(* Logix 5000 project; controller Drives_Line1 1756-L72 rev 20.13; software revision 20.04; part 10 of 21 *)
(* tags used below, declared in another part *)
   Bridle_01_FB_Count_Old : DINT;
   Bridle_01_Max_FBcounts : REAL;
   Bridle_01_SpdTrimMPS : REAL;
   Bridle_01_SpdTrimPct : REAL;
   Bridle_01a_RPMPerMPS : REAL;
   Bridle_01b_RPMPerMPS : REAL;
   Bridle_01c_RPMPerMPS : REAL;
   IO_State_Bridle_01a : INT;
   IO_State_Bridle_01b : INT;
   IO_State_Bridle_01c : INT;
   IO_State_Tmp_Bridle_01a : INT;
   IO_State_Tmp_Bridle_01b : INT;
   IO_State_Tmp_Bridle_01c : INT;
   zBridle_01_Ki_SpdTrim : REAL;
   zBridle_01_Kp_SpdTrim : REAL;
   zBridle_01_Max_rev : DINT;
   zBridle_01_MaxTrimSpdTrim : REAL;
   zBridle_01_MinTrimSpdTrim : REAL;
   zBridle_01b_EncRes : REAL;
   Bridle_01 : UDT_Bridle_3M;
   Bridle_01_FB_Diff : REAL;
   Bridle_01_FB_Update_Valid : BOOL;
   Bridle_01_Rev_mm : REAL;
   Bridle_01b_FBCounts_mm : REAL;
   EntryCtrl : UDT_Control_Zone;
   EntryStat : UDT_Status_Zone;
   LineCmd : UDT_Commands_Line;
   offst_pr_br1 : REAL;
   Out_Feedbacks : UDT_Fdbks;
   Out_Status : UDT_Status;
   TaskInterval_ms : DINT;
   TestConfig_Bridle_01a : UDT_Config_Bridle;
   TestConfig_Bridle_01b : UDT_Config_Bridle;
   TestConfig_Bridle_01c : UDT_Config_Bridle;
   voirmw : BOOL;
   zConfigFromMaster : BOOL;
   zPi : REAL;
   zSimulation : BOOL;
(* P14_Bridle_01, continued *)

ROUTINE R03_Drive_Interface   (* ladder *)
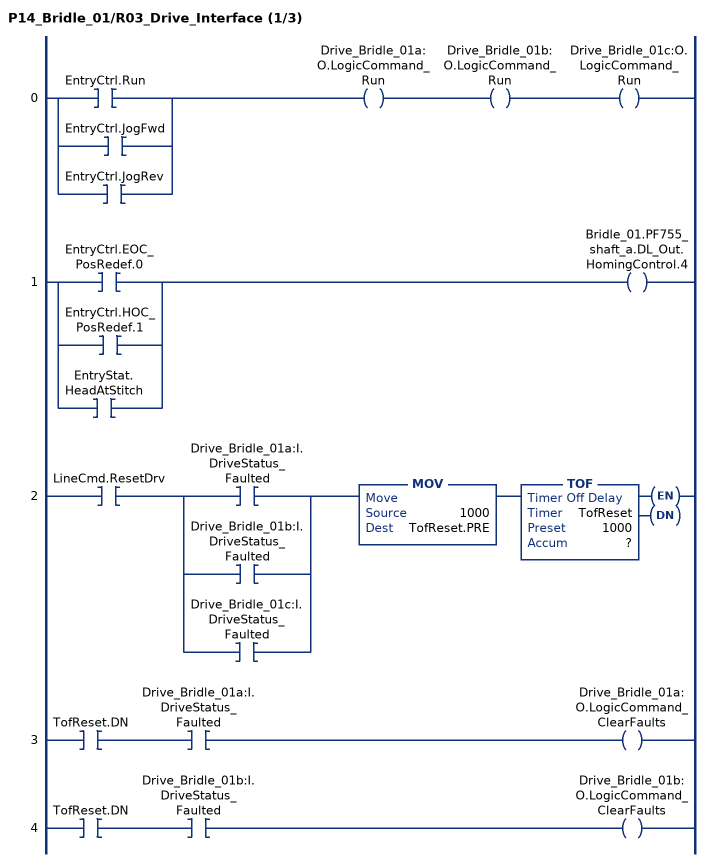
   0: [XIC(EntryCtrl.Run) ,XIC(EntryCtrl.JogFwd) ,XIC(EntryCtrl.JogRev) ]OTE(Drive_Bridle_01a:O.LogicCommand_Run)OTE(Drive_Bridle_01b:O.LogicCommand_Run)OTE(Drive_Bridle_01c:O.LogicCommand_Run);
   1: [XIC(EntryCtrl.EOC_PosRedef.0) ,XIC(EntryCtrl.HOC_PosRedef.1) ,XIC(EntryStat.HeadAtStitch) ]OTE(Bridle_01.PF755_shaft_a.DL_Out.HomingControl.4);
   2: XIC(LineCmd.ResetDrv)[XIC(Drive_Bridle_01a:I.DriveStatus_Faulted) ,XIC(Drive_Bridle_01b:I.DriveStatus_Faulted) ,XIC(Drive_Bridle_01c:I.DriveStatus_Faulted) ]MOV(1000,TofReset.PRE)TOF(TofReset,?,?);
   3: XIC(TofReset.DN)XIC(Drive_Bridle_01a:I.DriveStatus_Faulted)OTE(Drive_Bridle_01a:O.LogicCommand_ClearFaults);
   4: XIC(TofReset.DN)XIC(Drive_Bridle_01b:I.DriveStatus_Faulted)OTE(Drive_Bridle_01b:O.LogicCommand_ClearFaults);
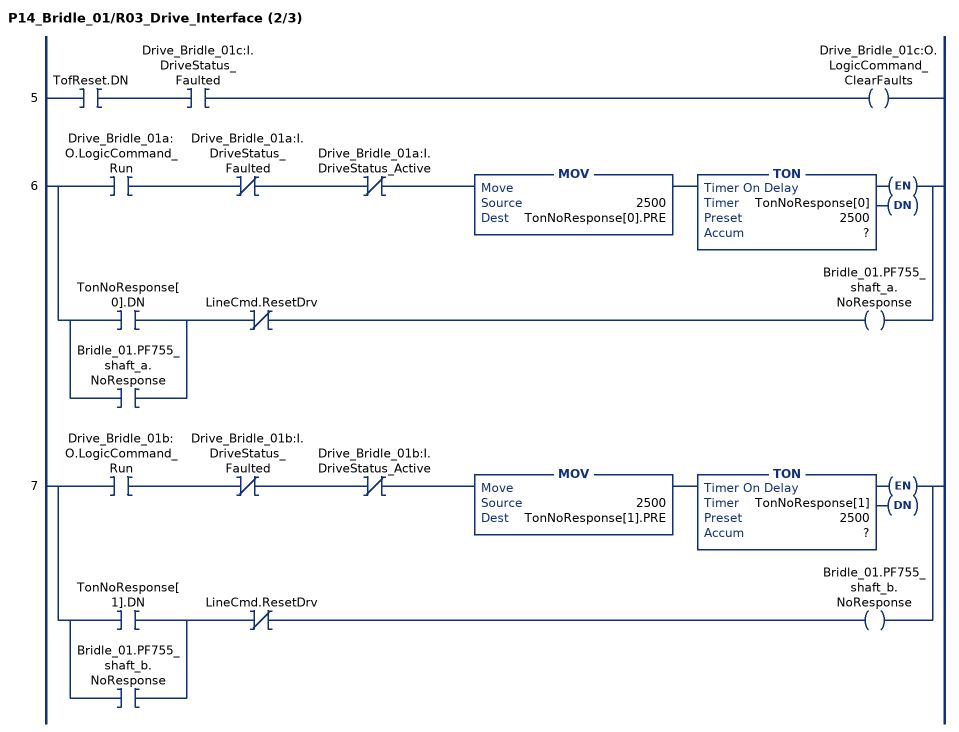
   5: XIC(TofReset.DN)XIC(Drive_Bridle_01c:I.DriveStatus_Faulted)OTE(Drive_Bridle_01c:O.LogicCommand_ClearFaults);
   6: [XIC(Drive_Bridle_01a:O.LogicCommand_Run) XIO(Drive_Bridle_01a:I.DriveStatus_Faulted) XIO(Drive_Bridle_01a:I.DriveStatus_Active) MOV(2500,TonNoResponse[0].PRE) TON(TonNoResponse[0],?,?) ,[XIC(TonNoResponse[0].DN) ,XIC(Bridle_01.PF755_shaft_a.NoResponse) ] XIO(LineCmd.ResetDrv) OTE(Bridle_01.PF755_shaft_a.NoResponse) ];
   7: [XIC(Drive_Bridle_01b:O.LogicCommand_Run) XIO(Drive_Bridle_01b:I.DriveStatus_Faulted) XIO(Drive_Bridle_01b:I.DriveStatus_Active) MOV(2500,TonNoResponse[1].PRE) TON(TonNoResponse[1],?,?) ,[XIC(TonNoResponse[1].DN) ,XIC(Bridle_01.PF755_shaft_b.NoResponse) ] XIO(LineCmd.ResetDrv) OTE(Bridle_01.PF755_shaft_b.NoResponse) ];
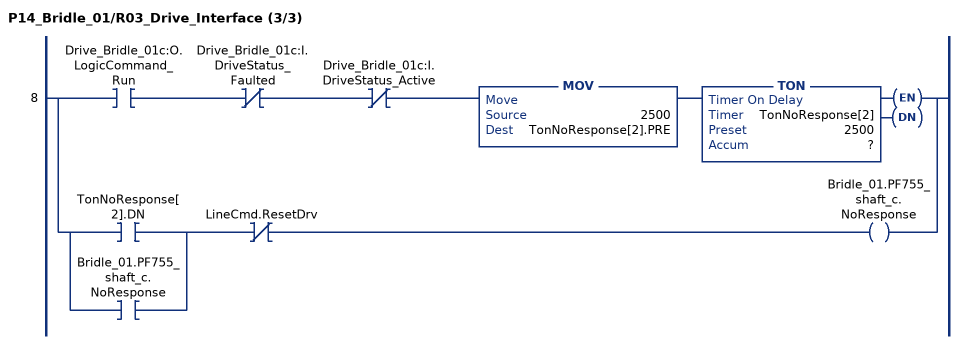
   8: [XIC(Drive_Bridle_01c:O.LogicCommand_Run) XIO(Drive_Bridle_01c:I.DriveStatus_Faulted) XIO(Drive_Bridle_01c:I.DriveStatus_Active) MOV(2500,TonNoResponse[2].PRE) TON(TonNoResponse[2],?,?) ,[XIC(TonNoResponse[2].DN) ,XIC(Bridle_01.PF755_shaft_c.NoResponse) ] XIO(LineCmd.ResetDrv) OTE(Bridle_01.PF755_shaft_c.NoResponse) ];
END_ROUTINE

ROUTINE R04_State   (* ladder *)
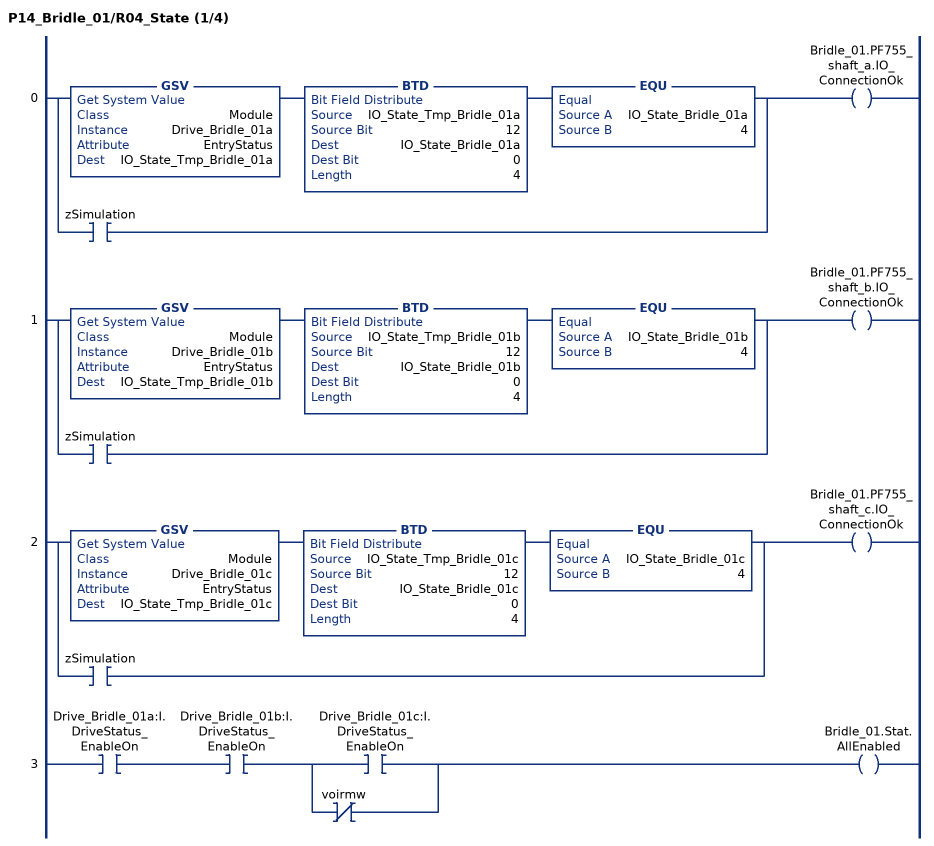
   0: [GSV(Module,Drive_Bridle_01a,EntryStatus,IO_State_Tmp_Bridle_01a) BTD(IO_State_Tmp_Bridle_01a,12,IO_State_Bridle_01a,0,4) EQU(IO_State_Bridle_01a,4) ,XIC(zSimulation) ]OTE(Bridle_01.PF755_shaft_a.IO_ConnectionOk);
   1: [GSV(Module,Drive_Bridle_01b,EntryStatus,IO_State_Tmp_Bridle_01b) BTD(IO_State_Tmp_Bridle_01b,12,IO_State_Bridle_01b,0,4) EQU(IO_State_Bridle_01b,4) ,XIC(zSimulation) ]OTE(Bridle_01.PF755_shaft_b.IO_ConnectionOk);
   2: [GSV(Module,Drive_Bridle_01c,EntryStatus,IO_State_Tmp_Bridle_01c) BTD(IO_State_Tmp_Bridle_01c,12,IO_State_Bridle_01c,0,4) EQU(IO_State_Bridle_01c,4) ,XIC(zSimulation) ]OTE(Bridle_01.PF755_shaft_c.IO_ConnectionOk);
   3: XIC(Drive_Bridle_01a:I.DriveStatus_EnableOn)XIC(Drive_Bridle_01b:I.DriveStatus_EnableOn)[XIC(Drive_Bridle_01c:I.DriveStatus_EnableOn) ,XIO(voirmw) ]OTE(Bridle_01.Stat.AllEnabled);
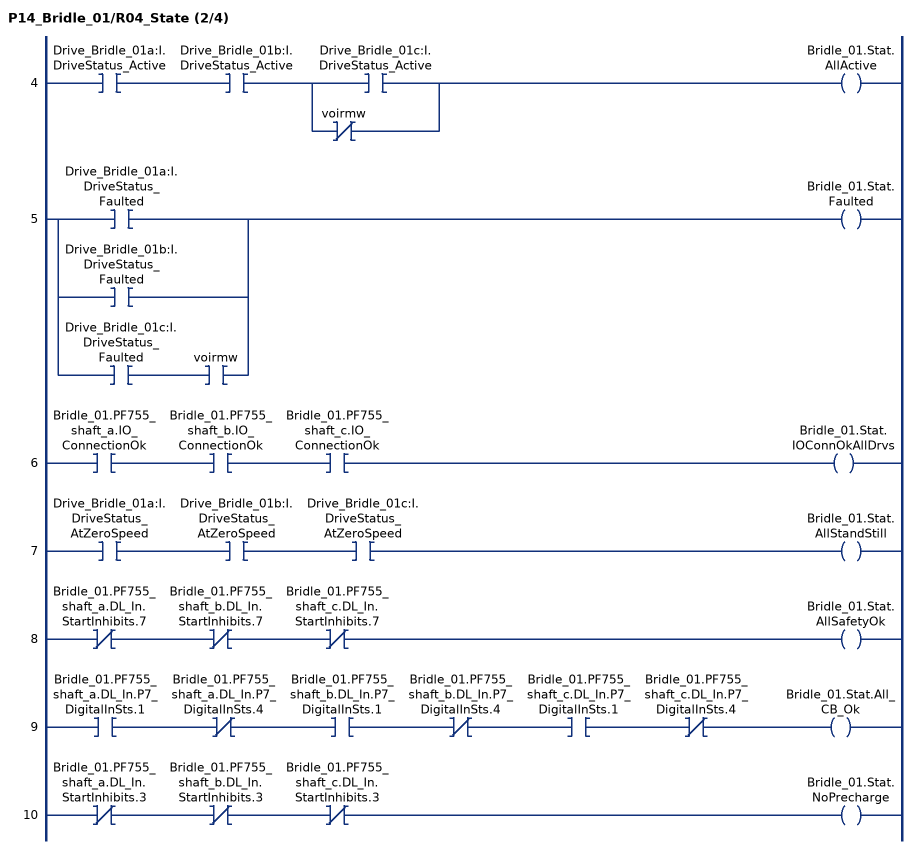
   4: XIC(Drive_Bridle_01a:I.DriveStatus_Active)XIC(Drive_Bridle_01b:I.DriveStatus_Active)[XIC(Drive_Bridle_01c:I.DriveStatus_Active) ,XIO(voirmw) ]OTE(Bridle_01.Stat.AllActive);
   5: [XIC(Drive_Bridle_01a:I.DriveStatus_Faulted) ,XIC(Drive_Bridle_01b:I.DriveStatus_Faulted) ,XIC(Drive_Bridle_01c:I.DriveStatus_Faulted) XIC(voirmw) ]OTE(Bridle_01.Stat.Faulted);
   6: XIC(Bridle_01.PF755_shaft_a.IO_ConnectionOk)XIC(Bridle_01.PF755_shaft_b.IO_ConnectionOk)XIC(Bridle_01.PF755_shaft_c.IO_ConnectionOk)OTE(Bridle_01.Stat.IOConnOkAllDrvs);
   7: XIC(Drive_Bridle_01a:I.DriveStatus_AtZeroSpeed)XIC(Drive_Bridle_01b:I.DriveStatus_AtZeroSpeed)XIC(Drive_Bridle_01c:I.DriveStatus_AtZeroSpeed)OTE(Bridle_01.Stat.AllStandStill);
   8: XIO(Bridle_01.PF755_shaft_a.DL_In.StartInhibits.7)XIO(Bridle_01.PF755_shaft_b.DL_In.StartInhibits.7)XIO(Bridle_01.PF755_shaft_c.DL_In.StartInhibits.7)OTE(Bridle_01.Stat.AllSafetyOk);
   9: XIC(Bridle_01.PF755_shaft_a.DL_In.P7_DigitalInSts.1)XIO(Bridle_01.PF755_shaft_a.DL_In.P7_DigitalInSts.4)XIC(Bridle_01.PF755_shaft_b.DL_In.P7_DigitalInSts.1)XIO(Bridle_01.PF755_shaft_b.DL_In.P7_DigitalInSts.4)XIC(Bridle_01.PF755_shaft_c.DL_In.P7_DigitalInSts.1)XIO(Bridle_01.PF755_shaft_c.DL_In.P7_DigitalInSts.4)OTE(Bridle_01.Stat.All_CB_Ok);
   10: XIO(Bridle_01.PF755_shaft_a.DL_In.StartInhibits.3)XIO(Bridle_01.PF755_shaft_b.DL_In.StartInhibits.3)XIO(Bridle_01.PF755_shaft_c.DL_In.StartInhibits.3)OTE(Bridle_01.Stat.NoPrecharge);
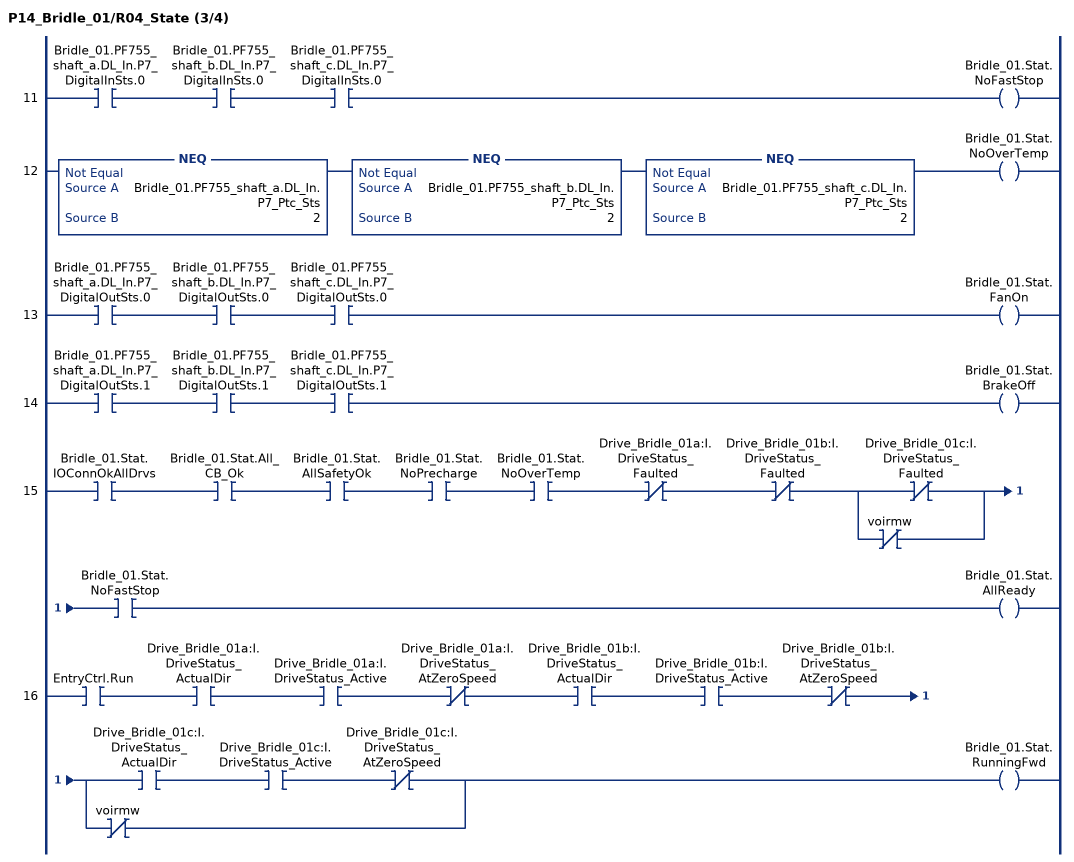
   11: XIC(Bridle_01.PF755_shaft_a.DL_In.P7_DigitalInSts.0)XIC(Bridle_01.PF755_shaft_b.DL_In.P7_DigitalInSts.0)XIC(Bridle_01.PF755_shaft_c.DL_In.P7_DigitalInSts.0)OTE(Bridle_01.Stat.NoFastStop);
   12: NEQ(Bridle_01.PF755_shaft_a.DL_In.P7_Ptc_Sts,2)NEQ(Bridle_01.PF755_shaft_b.DL_In.P7_Ptc_Sts,2)NEQ(Bridle_01.PF755_shaft_c.DL_In.P7_Ptc_Sts,2)OTE(Bridle_01.Stat.NoOverTemp);
   13: XIC(Bridle_01.PF755_shaft_a.DL_In.P7_DigitalOutSts.0)XIC(Bridle_01.PF755_shaft_b.DL_In.P7_DigitalOutSts.0)XIC(Bridle_01.PF755_shaft_c.DL_In.P7_DigitalOutSts.0)OTE(Bridle_01.Stat.FanOn);
   14: XIC(Bridle_01.PF755_shaft_a.DL_In.P7_DigitalOutSts.1)XIC(Bridle_01.PF755_shaft_b.DL_In.P7_DigitalOutSts.1)XIC(Bridle_01.PF755_shaft_c.DL_In.P7_DigitalOutSts.1)OTE(Bridle_01.Stat.BrakeOff);
   15: XIC(Bridle_01.Stat.IOConnOkAllDrvs)XIC(Bridle_01.Stat.All_CB_Ok)XIC(Bridle_01.Stat.AllSafetyOk)XIC(Bridle_01.Stat.NoPrecharge)XIC(Bridle_01.Stat.NoOverTemp)XIO(Drive_Bridle_01a:I.DriveStatus_Faulted)XIO(Drive_Bridle_01b:I.DriveStatus_Faulted)[XIO(Drive_Bridle_01c:I.DriveStatus_Faulted) ,XIO(voirmw) ]XIC(Bridle_01.Stat.NoFastStop)OTE(Bridle_01.Stat.AllReady);
   16: XIC(EntryCtrl.Run)XIC(Drive_Bridle_01a:I.DriveStatus_ActualDir)XIC(Drive_Bridle_01a:I.DriveStatus_Active)XIO(Drive_Bridle_01a:I.DriveStatus_AtZeroSpeed)XIC(Drive_Bridle_01b:I.DriveStatus_ActualDir)XIC(Drive_Bridle_01b:I.DriveStatus_Active)XIO(Drive_Bridle_01b:I.DriveStatus_AtZeroSpeed)[XIC(Drive_Bridle_01c:I.DriveStatus_ActualDir) XIC(Drive_Bridle_01c:I.DriveStatus_Active) XIO(Drive_Bridle_01c:I.DriveStatus_AtZeroSpeed) ,XIO(voirmw) ]OTE(Bridle_01.Stat.RunningFwd);
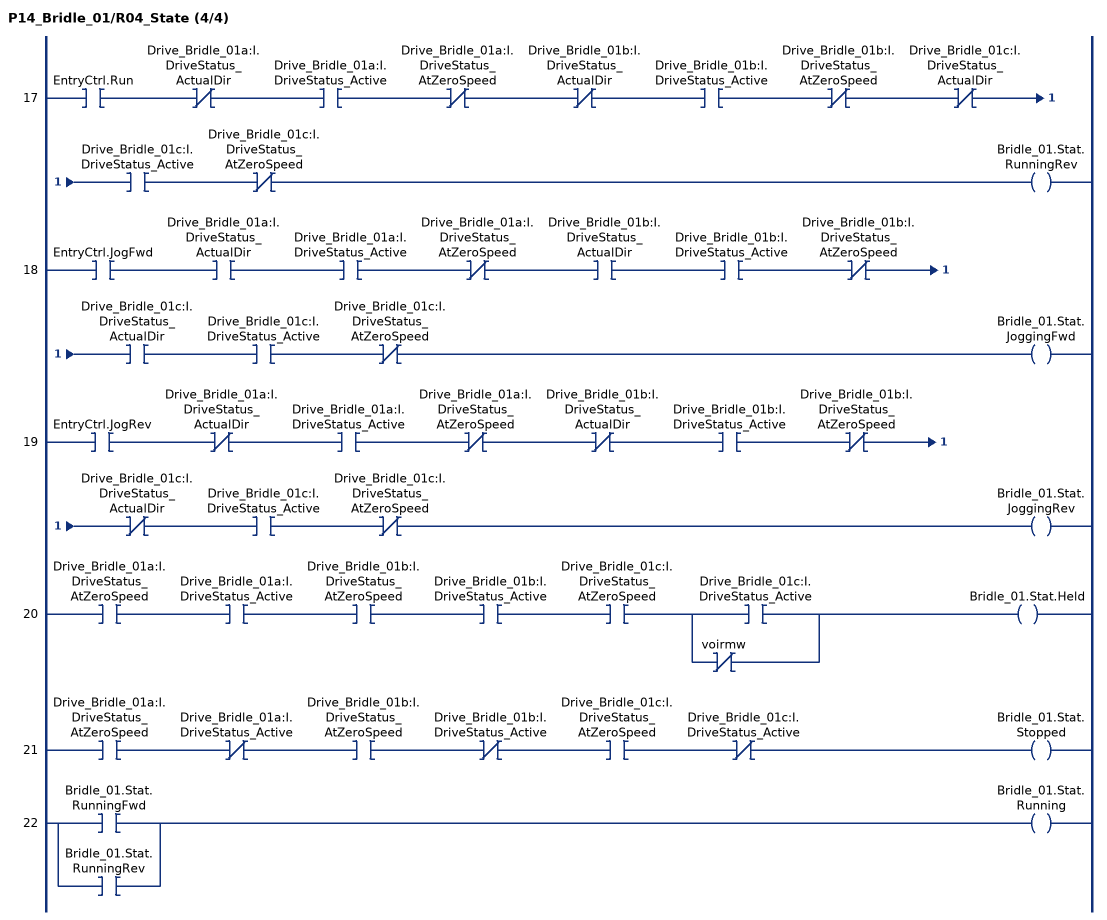
   17: XIC(EntryCtrl.Run)XIO(Drive_Bridle_01a:I.DriveStatus_ActualDir)XIC(Drive_Bridle_01a:I.DriveStatus_Active)XIO(Drive_Bridle_01a:I.DriveStatus_AtZeroSpeed)XIO(Drive_Bridle_01b:I.DriveStatus_ActualDir)XIC(Drive_Bridle_01b:I.DriveStatus_Active)XIO(Drive_Bridle_01b:I.DriveStatus_AtZeroSpeed)XIO(Drive_Bridle_01c:I.DriveStatus_ActualDir)XIC(Drive_Bridle_01c:I.DriveStatus_Active)XIO(Drive_Bridle_01c:I.DriveStatus_AtZeroSpeed)OTE(Bridle_01.Stat.RunningRev);
   18: XIC(EntryCtrl.JogFwd)XIC(Drive_Bridle_01a:I.DriveStatus_ActualDir)XIC(Drive_Bridle_01a:I.DriveStatus_Active)XIO(Drive_Bridle_01a:I.DriveStatus_AtZeroSpeed)XIC(Drive_Bridle_01b:I.DriveStatus_ActualDir)XIC(Drive_Bridle_01b:I.DriveStatus_Active)XIO(Drive_Bridle_01b:I.DriveStatus_AtZeroSpeed)XIC(Drive_Bridle_01c:I.DriveStatus_ActualDir)XIC(Drive_Bridle_01c:I.DriveStatus_Active)XIO(Drive_Bridle_01c:I.DriveStatus_AtZeroSpeed)OTE(Bridle_01.Stat.JoggingFwd);
   19: XIC(EntryCtrl.JogRev)XIO(Drive_Bridle_01a:I.DriveStatus_ActualDir)XIC(Drive_Bridle_01a:I.DriveStatus_Active)XIO(Drive_Bridle_01a:I.DriveStatus_AtZeroSpeed)XIO(Drive_Bridle_01b:I.DriveStatus_ActualDir)XIC(Drive_Bridle_01b:I.DriveStatus_Active)XIO(Drive_Bridle_01b:I.DriveStatus_AtZeroSpeed)XIO(Drive_Bridle_01c:I.DriveStatus_ActualDir)XIC(Drive_Bridle_01c:I.DriveStatus_Active)XIO(Drive_Bridle_01c:I.DriveStatus_AtZeroSpeed)OTE(Bridle_01.Stat.JoggingRev);
   20: XIC(Drive_Bridle_01a:I.DriveStatus_AtZeroSpeed)XIC(Drive_Bridle_01a:I.DriveStatus_Active)XIC(Drive_Bridle_01b:I.DriveStatus_AtZeroSpeed)XIC(Drive_Bridle_01b:I.DriveStatus_Active)XIC(Drive_Bridle_01c:I.DriveStatus_AtZeroSpeed)[XIC(Drive_Bridle_01c:I.DriveStatus_Active) ,XIO(voirmw) ]OTE(Bridle_01.Stat.Held);
   21: XIC(Drive_Bridle_01a:I.DriveStatus_AtZeroSpeed)XIO(Drive_Bridle_01a:I.DriveStatus_Active)XIC(Drive_Bridle_01b:I.DriveStatus_AtZeroSpeed)XIO(Drive_Bridle_01b:I.DriveStatus_Active)XIC(Drive_Bridle_01c:I.DriveStatus_AtZeroSpeed)XIO(Drive_Bridle_01c:I.DriveStatus_Active)OTE(Bridle_01.Stat.Stopped);
   22: [XIC(Bridle_01.Stat.RunningFwd) ,XIC(Bridle_01.Stat.RunningRev) ]OTE(Bridle_01.Stat.Running);
END_ROUTINE

ROUTINE R05_Control   (* ladder *)
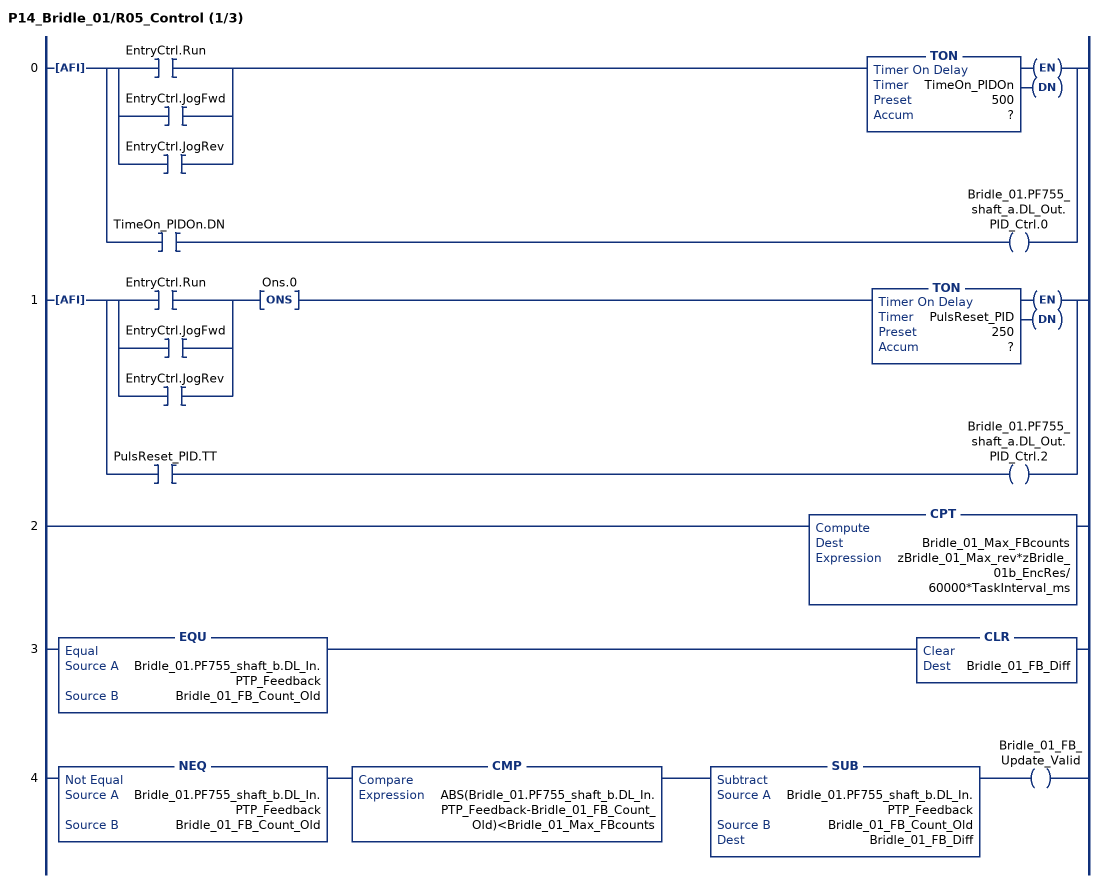
   0: AFI()[[XIC(EntryCtrl.Run) ,XIC(EntryCtrl.JogFwd) ,XIC(EntryCtrl.JogRev) ] TON(TimeOn_PIDOn,?,?) ,XIC(TimeOn_PIDOn.DN) OTE(Bridle_01.PF755_shaft_a.DL_Out.PID_Ctrl.0) ];
   1: AFI()[[XIC(EntryCtrl.Run) ,XIC(EntryCtrl.JogFwd) ,XIC(EntryCtrl.JogRev) ] ONS(Ons.0) TON(PulsReset_PID,?,?) ,XIC(PulsReset_PID.TT) OTE(Bridle_01.PF755_shaft_a.DL_Out.PID_Ctrl.2) ];
   2: CPT(Bridle_01_Max_FBcounts,zBridle_01_Max_rev*zBridle_01b_EncRes/60000*TaskInterval_ms);
   3: EQU(Bridle_01.PF755_shaft_b.DL_In.PTP_Feedback,Bridle_01_FB_Count_Old)CLR(Bridle_01_FB_Diff);
   4: NEQ(Bridle_01.PF755_shaft_b.DL_In.PTP_Feedback,Bridle_01_FB_Count_Old)CMP(ABS(Bridle_01.PF755_shaft_b.DL_In.PTP_Feedback-Bridle_01_FB_Count_Old)<Bridle_01_Max_FBcounts)SUB(Bridle_01.PF755_shaft_b.DL_In.PTP_Feedback,Bridle_01_FB_Count_Old,Bridle_01_FB_Diff)OTE(Bridle_01_FB_Update_Valid);
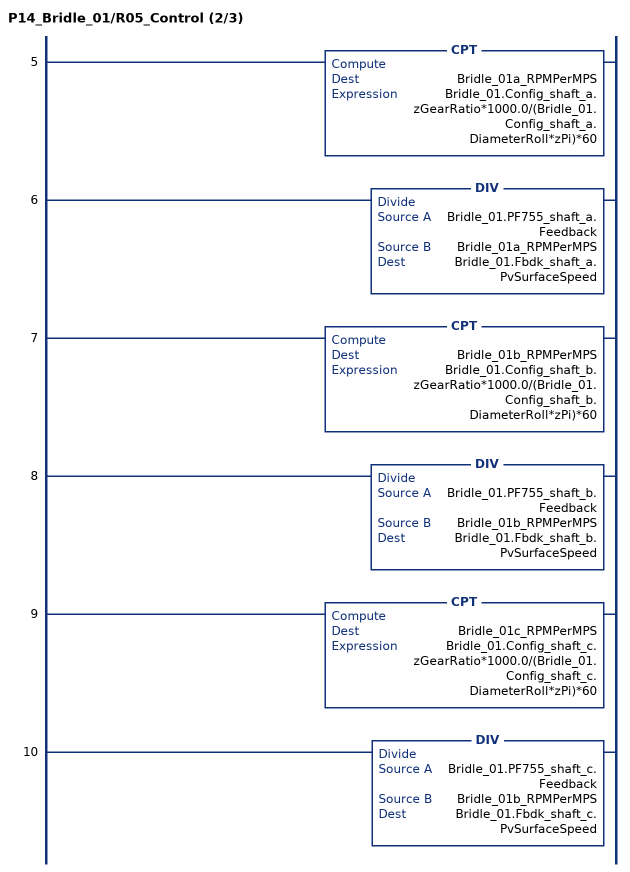
   5: CPT(Bridle_01a_RPMPerMPS,Bridle_01.Config_shaft_a.zGearRatio*1000.0/(Bridle_01.Config_shaft_a.DiameterRoll*zPi)*60);
   6: DIV(Bridle_01.PF755_shaft_a.Feedback,Bridle_01a_RPMPerMPS,Bridle_01.Fbdk_shaft_a.PvSurfaceSpeed);
   7: CPT(Bridle_01b_RPMPerMPS,Bridle_01.Config_shaft_b.zGearRatio*1000.0/(Bridle_01.Config_shaft_b.DiameterRoll*zPi)*60);
   8: DIV(Bridle_01.PF755_shaft_b.Feedback,Bridle_01b_RPMPerMPS,Bridle_01.Fbdk_shaft_b.PvSurfaceSpeed);
   9: CPT(Bridle_01c_RPMPerMPS,Bridle_01.Config_shaft_c.zGearRatio*1000.0/(Bridle_01.Config_shaft_c.DiameterRoll*zPi)*60);
   10: DIV(Bridle_01.PF755_shaft_c.Feedback,Bridle_01b_RPMPerMPS,Bridle_01.Fbdk_shaft_c.PvSurfaceSpeed);
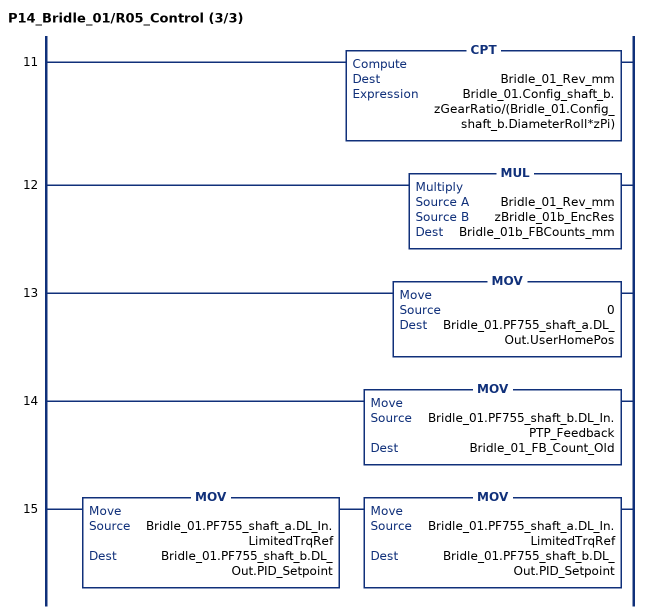
   11: CPT(Bridle_01_Rev_mm,Bridle_01.Config_shaft_b.zGearRatio/(Bridle_01.Config_shaft_b.DiameterRoll*zPi));
   12: MUL(Bridle_01_Rev_mm,zBridle_01b_EncRes,Bridle_01b_FBCounts_mm);
   13: MOV(0,Bridle_01.PF755_shaft_a.DL_Out.UserHomePos);
   14: MOV(Bridle_01.PF755_shaft_b.DL_In.PTP_Feedback,Bridle_01_FB_Count_Old);
   15: MOV(Bridle_01.PF755_shaft_a.DL_In.LimitedTrqRef,Bridle_01.PF755_shaft_b.DL_Out.PID_Setpoint)MOV(Bridle_01.PF755_shaft_a.DL_In.LimitedTrqRef,Bridle_01.PF755_shaft_b.DL_Out.PID_Setpoint);
END_ROUTINE

ROUTINE R11_LoadSharing   (* function block diagram *)
   SHEET 1   // Load sharing speed trim percentage
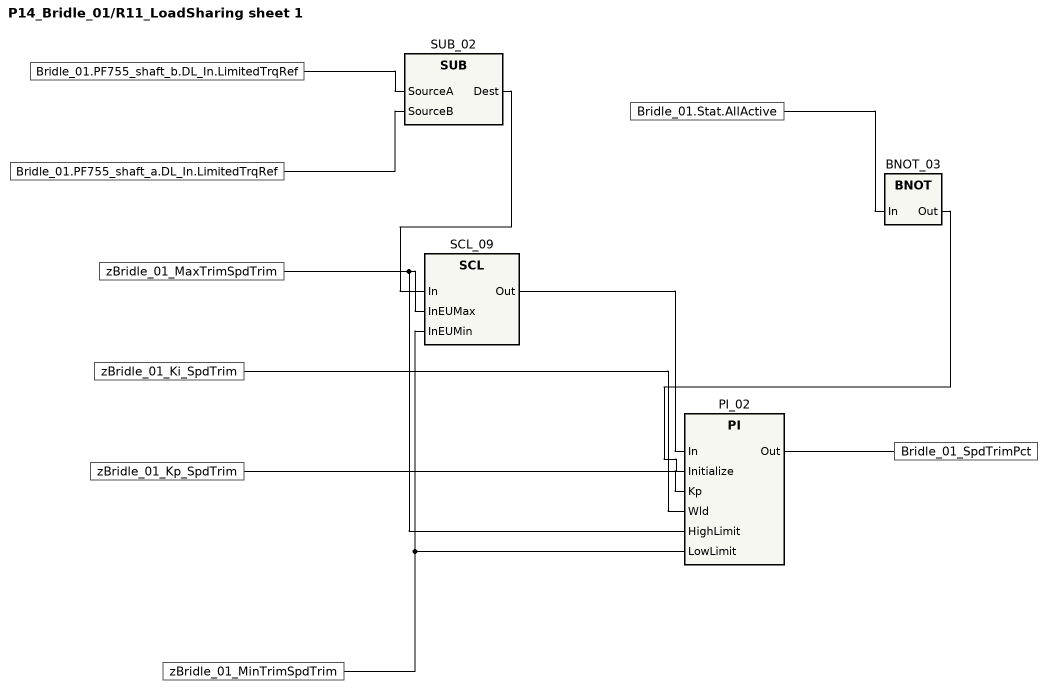
   SUB_02 : SUB(SourceA := Bridle_01.PF755_shaft_b.DL_In.LimitedTrqRef, SourceB := Bridle_01.PF755_shaft_a.DL_In.LimitedTrqRef);
   SCL_09 : SCL(In := SUB_02.Dest, InEUMax := zBridle_01_MaxTrimSpdTrim, InEUMin := zBridle_01_MinTrimSpdTrim);
   BNOT_03 : BNOT(In := Bridle_01.Stat.AllActive);
   PI_02 : PI(In := SCL_09.Out, Initialize := BNOT_03.Out, Kp := zBridle_01_Kp_SpdTrim, Wld := zBridle_01_Ki_SpdTrim, HighLimit := zBridle_01_MaxTrimSpdTrim, LowLimit := zBridle_01_MinTrimSpdTrim);
   Bridle_01_SpdTrimPct := PI_02.Out;
   SHEET 2   // Calculate speed trim mps
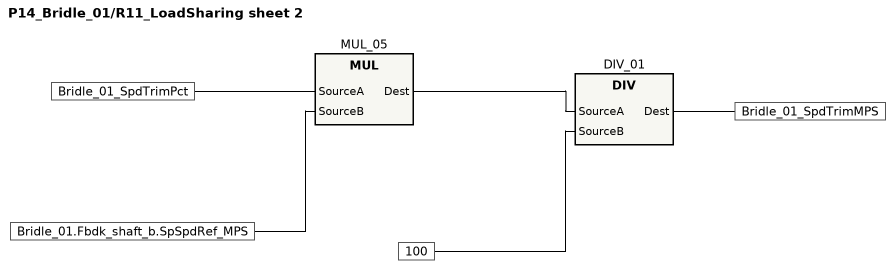
   MUL_05 : MUL(SourceA := Bridle_01_SpdTrimPct, SourceB := Bridle_01.Fbdk_shaft_b.SpSpdRef_MPS);
   DIV_01 : DIV(SourceA := MUL_05.Dest, SourceB := 100);
   Bridle_01_SpdTrimMPS := DIV_01.Dest;
END_ROUTINE

ROUTINE R12_DriveRef   (* function block diagram *)
   SHEET 1   // Final speed reference
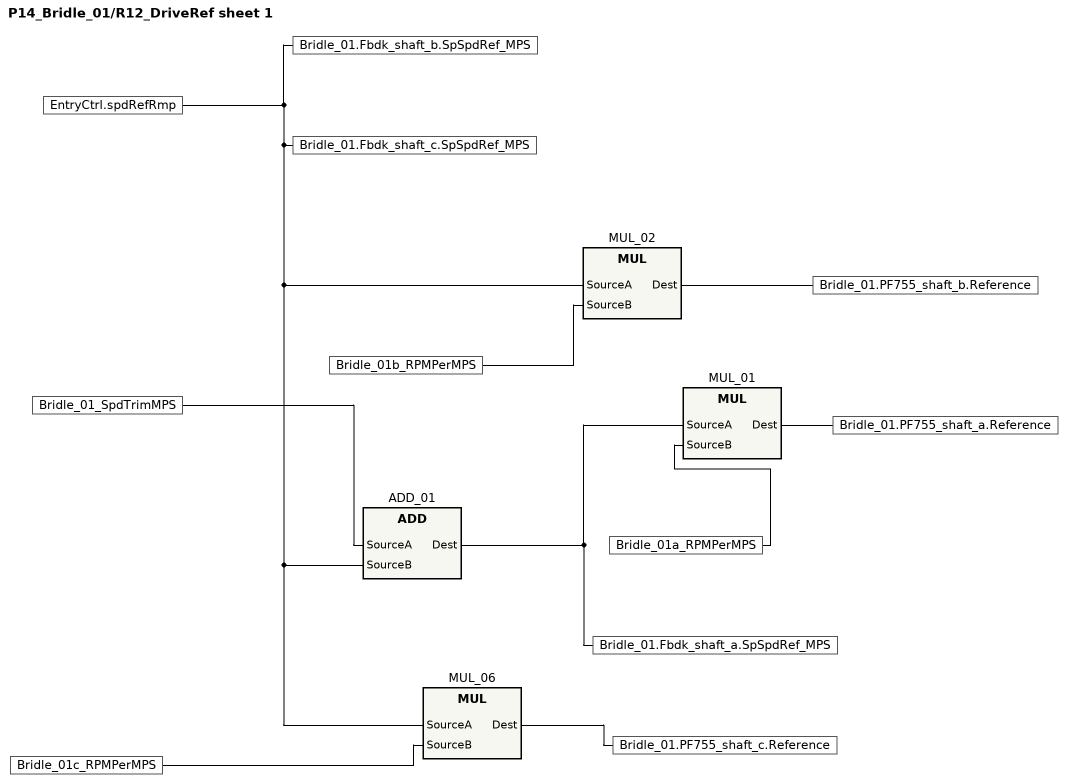
   Bridle_01.Fbdk_shaft_b.SpSpdRef_MPS := EntryCtrl.spdRefRmp;
   Bridle_01.Fbdk_shaft_c.SpSpdRef_MPS := EntryCtrl.spdRefRmp;
   ADD_01 : ADD(SourceA := Bridle_01_SpdTrimMPS, SourceB := EntryCtrl.spdRefRmp);
   MUL_06 : MUL(SourceA := EntryCtrl.spdRefRmp, SourceB := Bridle_01c_RPMPerMPS);
   MUL_02 : MUL(SourceA := EntryCtrl.spdRefRmp, SourceB := Bridle_01b_RPMPerMPS);
   Bridle_01.Fbdk_shaft_a.SpSpdRef_MPS := ADD_01.Dest;
   Bridle_01.PF755_shaft_c.Reference := MUL_06.Dest;
   MUL_01 : MUL(SourceA := ADD_01.Dest, SourceB := Bridle_01a_RPMPerMPS);
   Bridle_01.PF755_shaft_b.Reference := MUL_02.Dest;
   Bridle_01.PF755_shaft_a.Reference := MUL_01.Dest;
END_ROUTINE

ROUTINE R98_ToDrive   (* ladder *)
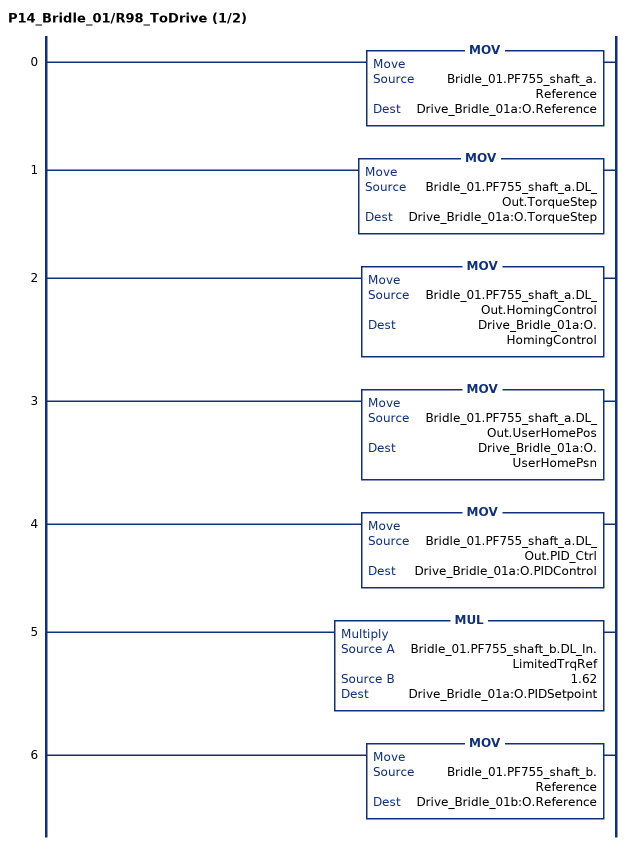
   0: MOV(Bridle_01.PF755_shaft_a.Reference,Drive_Bridle_01a:O.Reference);
   1: MOV(Bridle_01.PF755_shaft_a.DL_Out.TorqueStep,Drive_Bridle_01a:O.TorqueStep);
   2: MOV(Bridle_01.PF755_shaft_a.DL_Out.HomingControl,Drive_Bridle_01a:O.HomingControl);
   3: MOV(Bridle_01.PF755_shaft_a.DL_Out.UserHomePos,Drive_Bridle_01a:O.UserHomePsn);
   4: MOV(Bridle_01.PF755_shaft_a.DL_Out.PID_Ctrl,Drive_Bridle_01a:O.PIDControl);
   5: MUL(Bridle_01.PF755_shaft_b.DL_In.LimitedTrqRef,1.62,Drive_Bridle_01a:O.PIDSetpoint);
   6: MOV(Bridle_01.PF755_shaft_b.Reference,Drive_Bridle_01b:O.Reference);
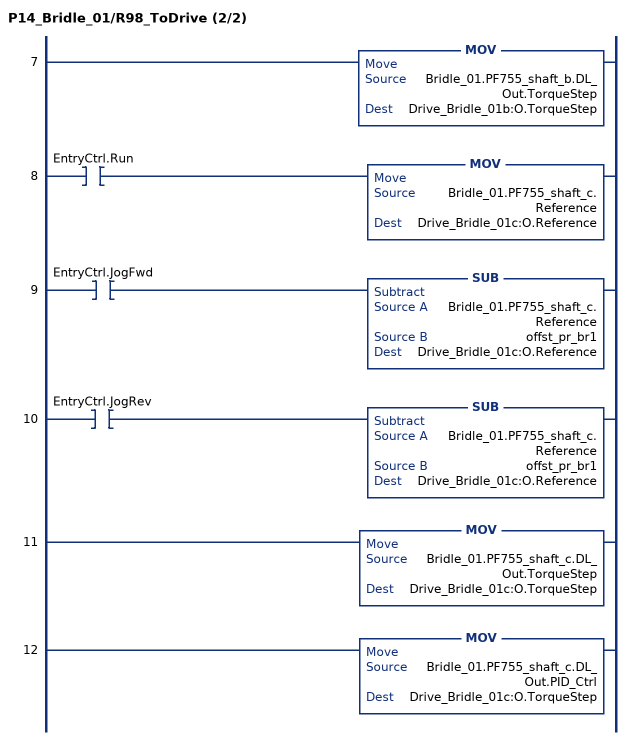
   7: MOV(Bridle_01.PF755_shaft_b.DL_Out.TorqueStep,Drive_Bridle_01b:O.TorqueStep);
   8: XIC(EntryCtrl.Run)MOV(Bridle_01.PF755_shaft_c.Reference,Drive_Bridle_01c:O.Reference);
   9: XIC(EntryCtrl.JogFwd)SUB(Bridle_01.PF755_shaft_c.Reference,offst_pr_br1,Drive_Bridle_01c:O.Reference);
   10: XIC(EntryCtrl.JogRev)SUB(Bridle_01.PF755_shaft_c.Reference,offst_pr_br1,Drive_Bridle_01c:O.Reference);
   11: MOV(Bridle_01.PF755_shaft_c.DL_Out.TorqueStep,Drive_Bridle_01c:O.TorqueStep);
   12: MOV(Bridle_01.PF755_shaft_c.DL_Out.PID_Ctrl,Drive_Bridle_01c:O.TorqueStep);
END_ROUTINE

ROUTINE R999_Test   (* ladder *)
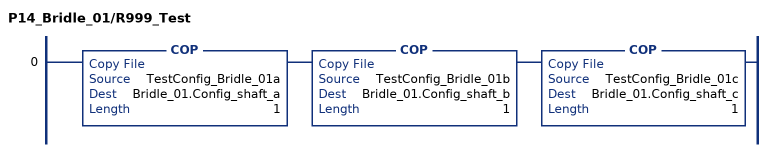
   0: COP(TestConfig_Bridle_01a,Bridle_01.Config_shaft_a,1)COP(TestConfig_Bridle_01b,Bridle_01.Config_shaft_b,1)COP(TestConfig_Bridle_01c,Bridle_01.Config_shaft_c,1);
END_ROUTINE

ROUTINE R99_To_Master   (* ladder *)
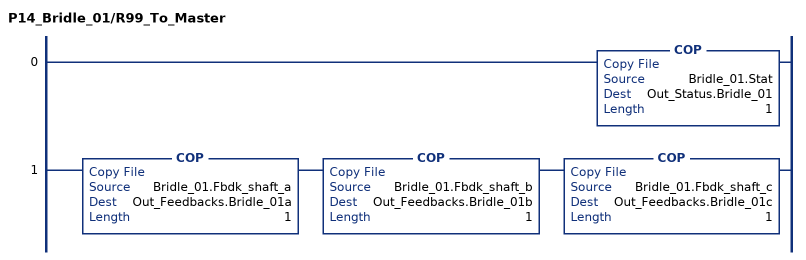
   0: COP(Bridle_01.Stat,Out_Status.Bridle_01,1);
   1: COP(Bridle_01.Fbdk_shaft_a,Out_Feedbacks.Bridle_01a,1)COP(Bridle_01.Fbdk_shaft_b,Out_Feedbacks.Bridle_01b,1)COP(Bridle_01.Fbdk_shaft_c,Out_Feedbacks.Bridle_01c,1);
END_ROUTINE
END_PROGRAM

PROGRAM P15_Bridle_02   (* main routine R00_Main *)
VAR
   ADD_01 : FBD_MATH := (SourceA := 0.00068994303, Dest := 0.00068994303);
   BAND_01 : FBD_BOOLEAN_AND := (In3 := 1, In4 := 1, In5 := 1, In6 := 1, In7 := 1, In8 := 1);
   BAND_03 : FBD_BOOLEAN_AND := (In3 := 1, In4 := 1, In5 := 1, In6 := 1, In7 := 1, In8 := 1);
   BNOT_01 : FBD_BOOLEAN_NOT := (Out := 1);
   BNOT_04 : FBD_BOOLEAN_NOT := (Out := 1);
   BNOT_06 : FBD_BOOLEAN_NOT := (Out := 1);
   Bridle_02_FB_Count_Old : DINT := -486222257;
   Bridle_02_Max_FBcounts : REAL := 5120.0;
   Bridle_02_SpdTrimMPS : REAL;
   Bridle_02_SpdTrimPct : REAL;
   Bridle_02a_RPMPerMPS : REAL := 6210.2964;
   Bridle_02b_RPMPerMPS : REAL := 6210.2964;
   DIV_01 : FBD_MATH := (SourceB := 100.0);
   EQU_01 : FBD_COMPARE := (SourceA := 0.083333336);
   IO_State_Bridle_02a : INT := 4;
   IO_State_Bridle_02b : INT := 4;
   IO_State_Tmp_Bridle_02a : INT := 16384;
   IO_State_Tmp_Bridle_02b : INT := 16384;
   MUL_01 : FBD_MATH := (SourceA := 0.00068994303, SourceB := 6210.2964, Dest := 4.284751);
   MUL_02 : FBD_MATH := (SourceA := 0.00068994303, SourceB := 6210.2964, Dest := 4.284751);
   MUL_05 : FBD_MATH := (SourceB := 0.00068994303);
   NEG_04 : FBD_MATH_ADVANCED := (Source := 0.083, Dest := -0.083);
   Ons : DINT;
   PI_02 : PROP_INT := (In := -2.3841858e-07, Initialize := 1, Kp := 0.8, Wld := 0.1, HighLimit := 2.5, LowLimit := -2.5, ShapeKpPlus := 1.0, ShapeKpMinus := 1.0, ShapeWldPlus := 1.0, ShapeWldMinus := 1.0, RTSTime := 1, DeltaT := 0.05);
   PulsReset_PID : TIMER := (PRE := 250);
   RLIM_01 : RATE_LIMITER := (In := 0.00068994303, IncRate := 0.5, DecRate := 0.5, RTSTime := 1, Out := 0.00068994303, DeltaT := 0.05);
   SCL_09 : SCALE := (InRawMax := 100.0, InRawMin := -100.0, InEUMax := 2.5, InEUMin := -2.5, Limiting := 1, Out := -2.3841858e-07);
   SCRV_01 : S_CURVE := (Initialize := 1, AbsAlgRamp := 1, AccelRate := 0.083, DecelRate := 0.083, JerkRate := 0.1, RTSTime := 1, DeltaT := 0.05);
   SSUM_03 : SELECTED_SUMMER := (In1 := 0.083, Gain1 := 1.0, In2 := -0.083, Gain2 := 1.0, Gain3 := 1.0, Select3 := 1, Gain4 := 1.0, Gain5 := 1.0, Gain6 := 1.0, Gain7 := 1.0, Gain8 := 1.0);
   SSUM_05 : SELECTED_SUMMER := (In1 := 0.00068994303, Gain1 := 1.0, Select1 := 1, Gain2 := 1.0, Gain3 := 1.0, Gain4 := 1.0, Gain5 := 1.0, Gain6 := 1.0, Gain7 := 1.0, Gain8 := 1.0, Out := 0.00068994303);
   SUB_02 : FBD_MATH;
   TimeOn_PIDOn : TIMER := (PRE := 500);
   TofReset : TIMER := (PRE := 1000, ACC := 1000);
   TonNoResponse : TIMER[3] := ([0].PRE := 2500, [1].PRE := 2500, [2].PRE := 2500, [2].ACC := 2500, [2].EN := 1, [2].DN := 1);
   TonRefOn : TIMER := (PRE := 500);
   zBridle_02_Ki_SpdTrim : REAL := 0.1;
   zBridle_02_Kp_SpdTrim : REAL := 0.8;
   zBridle_02_Max_rev : DINT := 1500;
   zBridle_02_MaxAccDec : REAL := 0.5;
   zBridle_02_MaxTrimSpdTrim : REAL := 2.5;
   zBridle_02_MinTrimSpdTrim : REAL := -2.5;
   zBridle_02b_EncRes : DINT := 4096;
END_VAR

ROUTINE R00_Main   (* ladder *)
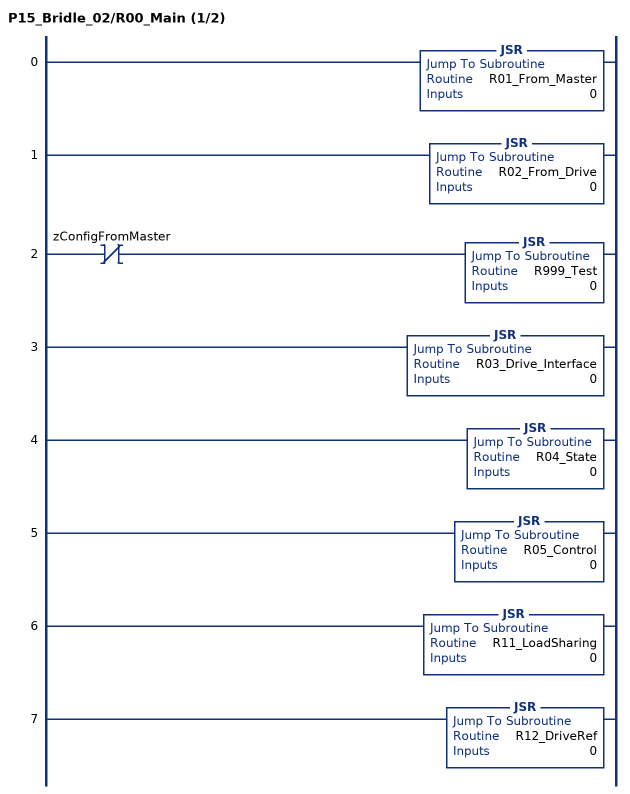
   0: JSR(R01_From_Master,0);
   1: JSR(R02_From_Drive,0);
   2: XIO(zConfigFromMaster)JSR(R999_Test,0);
   3: JSR(R03_Drive_Interface,0);
   4: JSR(R04_State,0);
   5: JSR(R05_Control,0);
   6: JSR(R11_LoadSharing,0);
   7: JSR(R12_DriveRef,0);
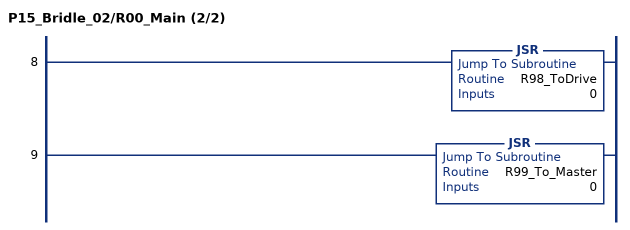
   8: JSR(R98_ToDrive,0);
   9: JSR(R99_To_Master,0);
END_ROUTINE
